// TIA Portal V19 export
TYPE "IPC_Msg_Generico"
   STRUCT
      Id : DInt;   // Identificativo progressivo univoco del messaggio (0 = cella vuota)
      timestamp : String;   // Timestamp evento formato ISO: YYYY-MM-DD HH:MM:SS.mmm
      topic : UDInt;   // Categoria/argomento del log per filtering e routing
      payLoad : String;   // Descrizione dettagliata dell'evento
   END_STRUCT;
END_TYPE
